// SIMATIC S7-200 project (STEP 7-Micro/WIN), CPU 226 CN REL 02.01

ORGANIZATION_BLOCK 程序块:OB1
TITLE=程序注释
BEGIN
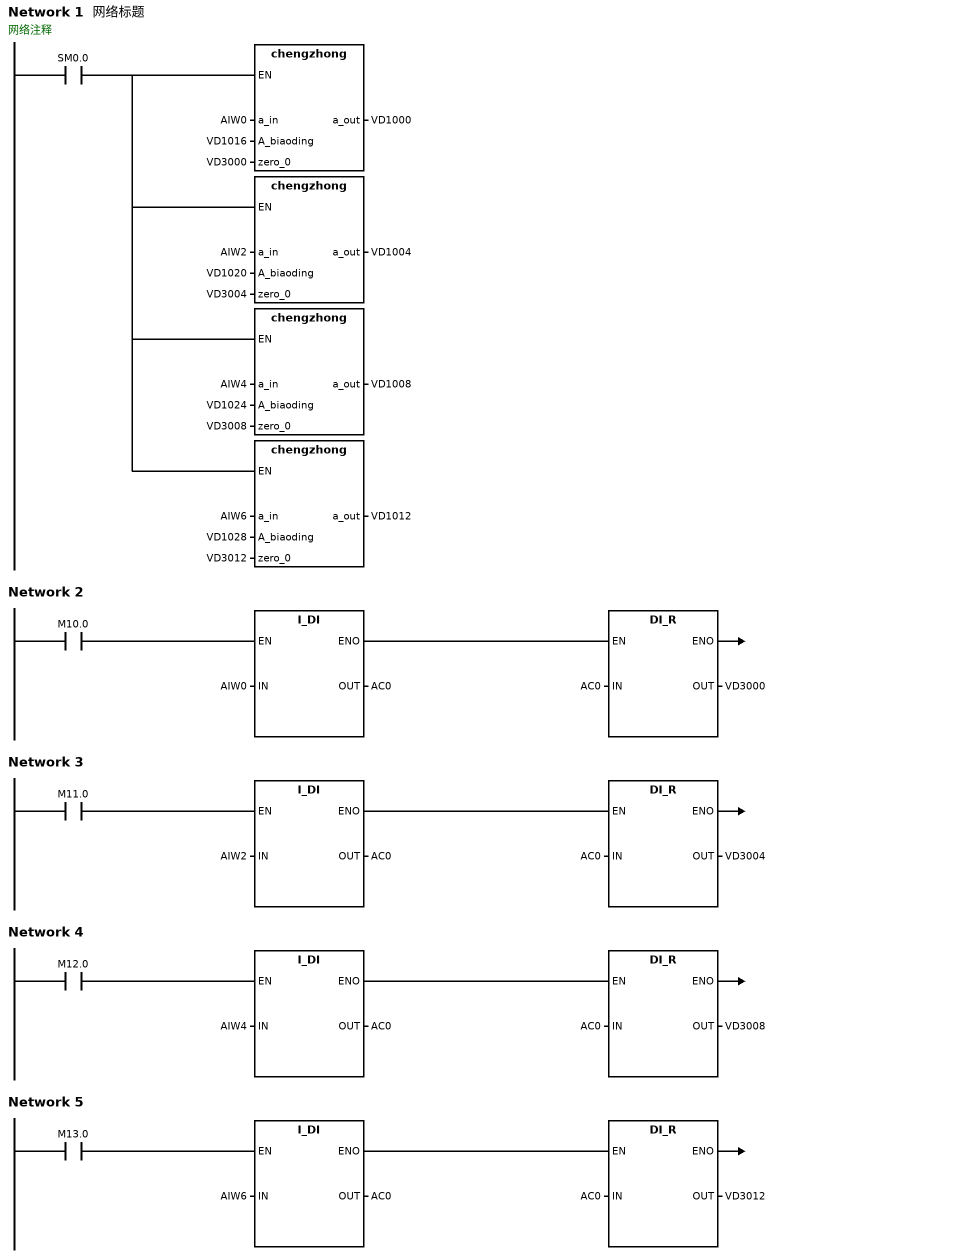
Network 1 // 网络标题
// 网络注释
LD     SM0.0
CALL   chengzhong:SBR0, AIW0, VD1016, VD3000, VD1000
CALL   chengzhong:SBR0, AIW2, VD1020, VD3004, VD1004
CALL   chengzhong:SBR0, AIW4, VD1024, VD3008, VD1008
CALL   chengzhong:SBR0, AIW6, VD1028, VD3012, VD1012
Network 2
LD     M10.0
ITD    AIW0, AC0
AENO
DTR    AC0, VD3000
Network 3
LD     M11.0
ITD    AIW2, AC0
AENO
DTR    AC0, VD3004
Network 4
LD     M12.0
ITD    AIW4, AC0
AENO
DTR    AC0, VD3008
Network 5
LD     M13.0
ITD    AIW6, AC0
AENO
DTR    AC0, VD3012
END_ORGANIZATION_BLOCK

SUBROUTINE_BLOCK chengzhong:SBR0
TITLE=子程序注释
VAR_INPUT
a_in:WORD;	// LW0 
A_biaoding:REAL;	// LD2 
zero_0:REAL;	// LD6 
END_VAR
VAR_OUTPUT
a_out:REAL;	// LD10 
END_VAR
BEGIN
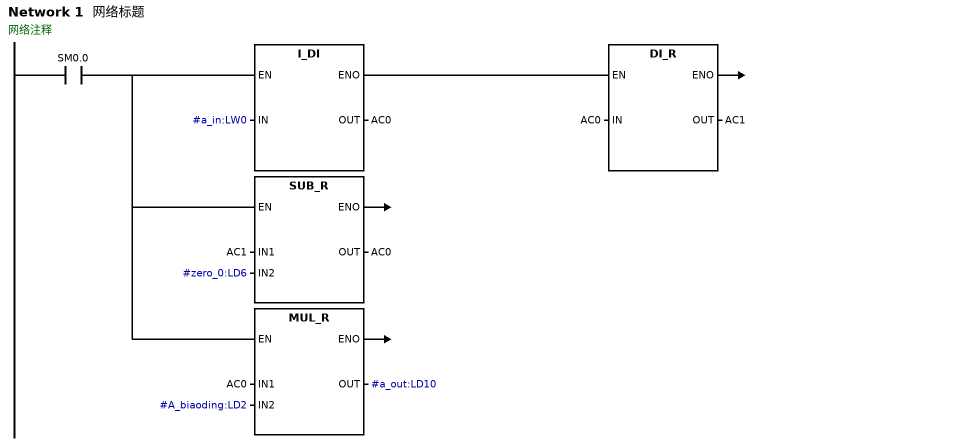
Network 1 // 网络标题
// 网络注释
LD     SM0.0
LPS
ITD    #a_in:LW0, AC0
AENO
DTR    AC0, AC1
LRD
MOVR   AC1, AC0
-R     #zero_0:LD6, AC0
LPP
MOVR   AC0, #a_out:LD10
*R     #A_biaoding:LD2, #a_out:LD10
END_SUBROUTINE_BLOCK

SUBROUTINE_BLOCK SBR_1:SBR1
TITLE=子程序注释
VAR_INPUT
zero_key:BOOL;	// L0.0 
aa_in:WORD;	// LW1 
END_VAR
VAR_OUTPUT
zero_out:REAL;	// LD3 
END_VAR
BEGIN
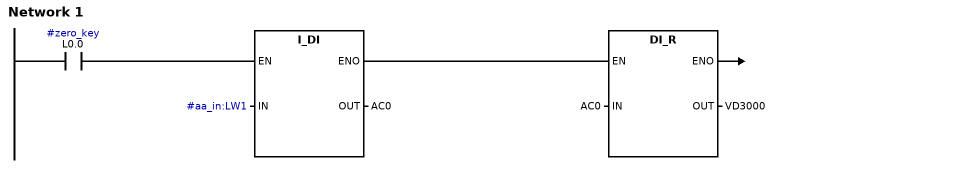
Network 1
LD     #zero_key:L0.0
ITD    #aa_in:LW1, AC0
AENO
DTR    AC0, VD3000
Network 2 // 网络标题
// 网络注释
END_SUBROUTINE_BLOCK
